// TwinCAT 3 PLC project SPS
// Company: mbc engineering GmbH
// ProgramVersion: 3.1.4022.2
// libraries:
//   Tc2_Standard, * (Beckhoff Automation GmbH)
//   Tc2_System, * (Beckhoff Automation GmbH)
//   Tc3_Module, * (Beckhoff Automation GmbH)
//   MBC TC3 PCS Library,newest,mbc engineering GmbH
// project tree:
//   DUTs/ ST_AddCommand.TcDUT, ST_AddCommandIn.TcDUT, ST_AddCommandOut.TcDUT, ST_BasicCommand.TcDUT, ST_CommandControl.TcDUT
//   GVLs/ Commands.TcGVL
//   / PlcTask.TcTTO
//   POUs/Commands/ AddCommand.TcPOU, DelayedAddCommand.TcPOU, StartCommand.TcPOU
//   POUs/ MAIN.TcPOU

CONFIGURATION SPS
    RESOURCE PLC ON TwinCAT3
        TASK PlcTask(INTERVAL := T#10ms, PRIORITY := 20);
        PROGRAM MAIN WITH PlcTask : MAIN;
    END_RESOURCE
END_CONFIGURATION

// ---- DUTs/ST_AddCommand.TcDUT
TYPE ST_AddCommand EXTENDS ST_BasicCommand :
STRUCT
	stArgsIn		: ST_AddCommandIn;
	stArgsOut		: ST_AddCommandOut;
END_STRUCT
END_TYPE

// ---- DUTs/ST_AddCommandIn.TcDUT
TYPE ST_AddCommandIn :
STRUCT
	a		: REAL;
	b		: REAL;
END_STRUCT
END_TYPE

// ---- DUTs/ST_AddCommandOut.TcDUT
TYPE ST_AddCommandOut :
STRUCT
	result		: REAL;
END_STRUCT
END_TYPE

// ---- DUTs/ST_BasicCommand.TcDUT
TYPE ST_BasicCommand :
STRUCT
	stCmd		: ST_CommandControl;
END_STRUCT
END_TYPE

// ---- DUTs/ST_CommandControl.TcDUT
TYPE ST_CommandControl :
STRUCT
	bExecute		: BOOL;		// Wird von PCS gesetzt um die Ausführung zu starten; zurücksetzen bricht die Ausführung ab
	bBusy			: BOOL;		// Anzeige, dass die Ausführung in der SPS läuft
	nResultCode		: UINT;		// Resultat der letzten Ausführung (bExecute & bBusy = FALSE)
END_STRUCT
END_TYPE

// ---- GVLs/Commands.TcGVL
{attribute 'qualified_only'}
VAR_GLOBAL
	stAddCommand		: ST_AddCommand;
	stAddLongCommand	: ST_AddCommand;
	
	
	AddCommand1			: AddCommand 			:= (Val1 := 3, Val2 := 2);
	DelayedAddCommand1	: DelayedAddCommand 	:= (Val1 := 4, Val2 := 5);
	StartCommand1		: StartCommand;		
END_VAR

// ---- POUs/MAIN.TcPOU
PROGRAM MAIN
VAR
	fbLongRunning		: TON := (PT:=T#4s);
	counter				: UINT;
	fbTof: TOF;
END_VAR

Commands.StartCommand1.Refresh();

fbTof(
	IN := Commands.StartCommand1.Q,
	PT := T#1S);
	





counter := counter + 1;


// Function variant
Commands.AddCommand1.Refresh();
Commands.DelayedAddCommand1.Refresh();

// Strukture variant
IF Commands.stAddCommand.stCmd.bExecute THEN
	Commands.stAddCommand.stArgsOut.result :=
		Commands.stAddCommand.stArgsIn.a + Commands.stAddCommand.stArgsIn.b;
	Commands.stAddCommand.stCmd.nResultCode := 0;
	Commands.stAddCommand.stCmd.bBusy := Commands.stAddCommand.stCmd.bExecute := FALSE;
END_IF

// Länger gehendes Kommando
IF Commands.stAddLongCommand.stCmd.bExecute THEN
	Commands.stAddLongCommand.stCmd.bBusy := TRUE;
END_IF

IF NOT Commands.stAddLongCommand.stCmd.bExecute AND Commands.stAddLongCommand.stCmd.bBusy THEN
	Commands.stAddLongCommand.stCmd.bBusy := FALSE;
	Commands.stAddLongCommand.stCmd.nResultCode := 5;
END_IF

fbLongRunning(IN:=Commands.stAddLongCommand.stCmd.bBusy);

IF fbLongRunning.Q THEN
	Commands.stAddLongCommand.stArgsOut.result :=
		Commands.stAddLongCommand.stArgsIn.a + Commands.stAddLongCommand.stArgsIn.b;
	Commands.stAddLongCommand.stCmd.nResultCode := 0;
	Commands.stAddLongCommand.stCmd.bBusy := Commands.stAddLongCommand.stCmd.bExecute := FALSE;	
END_IF

END_PROGRAM

// ---- POUs/Commands/AddCommand.TcPOU
FUNCTION_BLOCK AddCommand EXTENDS CommandBase
VAR_INPUT
	Val1 : REAL;
	Val2 : REAL;
END_VAR
VAR_OUTPUT 
	// The result of the addition command
	Result : REAL;	
END_VAR
VAR
END_VAR

// OO-Class 
;

METHOD PROTECTED Task : BOOL
VAR_INPUT
	Init 	: BOOL;		// True the first time the Task is called after Execute is started
END_VAR
Result := Val1 + Val2;

// Task comlete;
Task := SUPER^.Task(Init);;
END_METHOD

END_FUNCTION_BLOCK

// ---- POUs/Commands/DelayedAddCommand.TcPOU
FUNCTION_BLOCK DelayedAddCommand EXTENDS AddCommand
VAR
	_tonDelay		: TON := (PT:=T#4s);
END_VAR

METHOD PUBLIC Abort
SUPER^.Abort();

// Reset Input for next start
_tonDelay(IN:=stHandshake.bBusy);
END_METHOD

METHOD PROTECTED CalculateProgress
IF stHandshake.nResultCode = E_CommandResultCode.Done THEN
	stHandshake.nProgress := 100;
ELSE
	stHandshake.nProgress := REAL_TO_BYTE(100.0 / TIME_TO_REAL(_tonDelay.PT) * TIME_TO_REAL(_tonDelay.ET));
END_IF
END_METHOD

METHOD PROTECTED Done
VAR_INPUT
	nResultCode		: UINT;
END_VAR
SUPER^.Done(nResultCode);

// Reset Input for next start
_tonDelay(IN:=stHandshake.bBusy);
END_METHOD

METHOD PROTECTED Task : BOOL
_tonDelay(IN:=stHandshake.bBusy);

IF _tonDelay.Q THEN
	// Execute base Task in AddCommand for Addition
	Task := SUPER^.Task();
END_IF
END_METHOD

END_FUNCTION_BLOCK

// ---- POUs/Commands/StartCommand.TcPOU
FUNCTION_BLOCK PUBLIC StartCommand EXTENDS CommandBase
VAR_INPUT
END_VAR
VAR_OUTPUT	
	Q : BOOL;
END_VAR
VAR
END_VAR

METHOD PROTECTED Task : BOOL
VAR_INPUT
	Init 	: BOOL;		// True the first time the Task is called after Execute is started
END_VAR
IF (NOT Init AND Q) THEN
	// Task comlete;
	Task := SUPER^.Task(Init);;
END_IF

// set init
Q := Init;
END_METHOD

END_FUNCTION_BLOCK
